INTERFACE ITcoKeyNormalSevice

PROPERTY KeyInNormal : BOOL
GET
END_GET
END_PROPERTY

PROPERTY KeyInService : BOOL
GET
END_GET
END_PROPERTY

END_INTERFACE

(* stored: Version 1.1.0.1
   Itf ITcoKeyNormalSevice: Id {4d3292d3-2bbd-4847-b304-f02ce9ea0edc}
   Property KeyInNormal: Id {c06bb553-1c28-4af4-8591-1c745d4847b9}
   Get Get: Id {a652bfaa-502b-4c47-a7ca-c910d577b3e0}
   Property KeyInService: Id {1ac2d69d-31f4-46d6-ae52-dea8b0f4da43}
   Get Get: Id {52ba5769-e7f4-4845-aef5-40ef3d505173} *)
